PROGRAM MAIN
VAR
	_tcc : tcc;

END_VAR

//_tcc.Run();

END_PROGRAM

(* stored: Version 1.1.0.1, ProductVersion 3.1.4024.9
   POU MAIN: Id {18959407-38bc-0c60-272f-7f97dd416956}, SpecialFunc None *)
